/// Enumeration of all axis drives.
TYPE E_DigitalOutput :
(
	eDigitalOutput_OutletBelt					:= 0 ,

	
	// IMPORTANT: last entry
	eDigitalOutput_max
);
END_TYPE

(* stored: Version 1.1.0.1, ProductVersion 3.1.4022.10
   DUT E_DigitalOutput: Id {fef308ee-866e-4f15-92ce-925fe16852d6} *)
